% RSLogix 500 project PROCESO.RSS, saved by version 8.40.00.08 %
PROJECT "UNTITLED"    % processor: MicroLogix 1500 %

PROGRAM FILES
  LAD 2   34 rungs

DATA FILES
  O0 OUTPUT  6 elements
  I1 INPUT  5 elements
  S2 STATUS  66 elements
  B3 BINARY  1 elements
  T4 TIMER  10 elements
  C5 COUNTER  1 elements
  R6 CONTROL  1 elements
  N7 INTEGER  1 elements
  F8 FLOAT  1 elements

LADDER 2
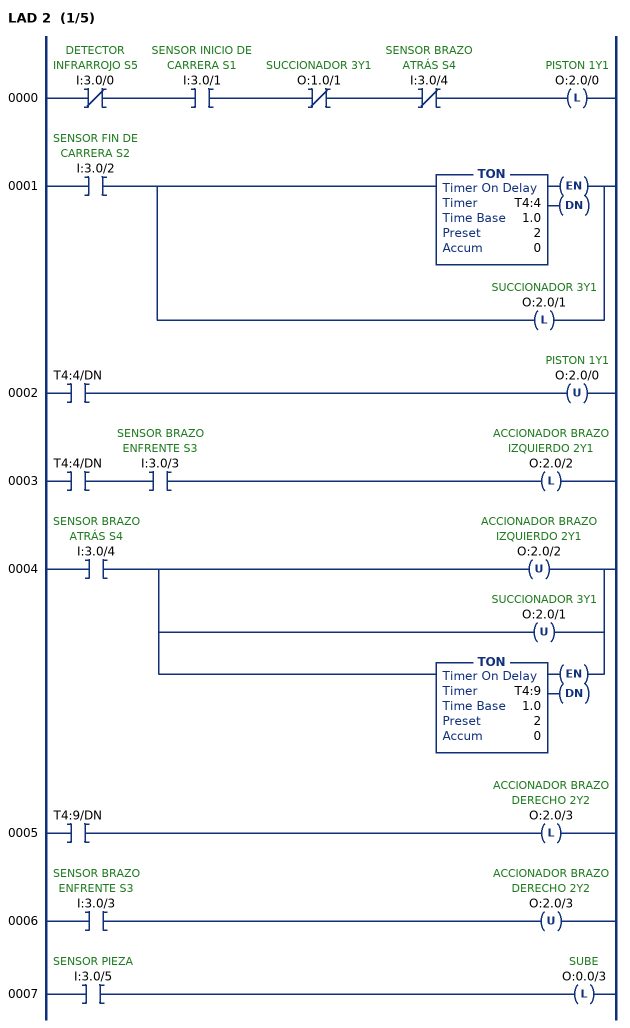
% Rung: 0 %
SOR XIO I:3.0/0 XIC I:3.0/1 XIO O:1.0/1 XIO I:3.0/4 OTL O:2.0/0 EOR
%   I:3.0/0  "DETECTOR INFRARROJO S5" %
%   I:3.0/1  "SENSOR INICIO DE CARRERA S1" %
%   O:1.0/1  "SUCCIONADOR 3Y1" %
%   I:3.0/4  "SENSOR BRAZO ATRÁS S4" %
%   O:2.0/0  "PISTON 1Y1" %
% Rung: 1 %
SOR XIC I:3.0/2 BST TON T4:4 1.0 2 0 NXB OTL O:2.0/1 BND EOR
%   I:3.0/2  "SENSOR FIN DE CARRERA S2" %
%   O:2.0/1  "SUCCIONADOR 3Y1" %
% Rung: 2 %
SOR XIC T4:4/DN OTU O:2.0/0 EOR
%   O:2.0/0  "PISTON 1Y1" %
% Rung: 3 %
SOR XIC T4:4/DN XIC I:3.0/3 OTL O:2.0/2 EOR
%   I:3.0/3  "SENSOR BRAZO ENFRENTE S3" %
%   O:2.0/2  "ACCIONADOR BRAZO IZQUIERDO 2Y1" %
% Rung: 4 %
SOR XIC I:3.0/4 BST OTU O:2.0/2 NXB BST OTU O:2.0/1 NXB TON T4:9 1.0 2 0 BND BND EOR
%   I:3.0/4  "SENSOR BRAZO ATRÁS S4" %
%   O:2.0/2  "ACCIONADOR BRAZO IZQUIERDO 2Y1" %
%   O:2.0/1  "SUCCIONADOR 3Y1" %
% Rung: 5 %
SOR XIC T4:9/DN OTL O:2.0/3 EOR
%   O:2.0/3  "ACCIONADOR BRAZO DERECHO 2Y2" %
% Rung: 6 %
SOR XIC I:3.0/3 OTU O:2.0/3 EOR
%   I:3.0/3  "SENSOR BRAZO ENFRENTE S3" %
%   O:2.0/3  "ACCIONADOR BRAZO DERECHO 2Y2" %
% Rung: 7 %
SOR XIC I:3.0/5 OTL O:0.0/3 EOR
%   I:3.0/5  "SENSOR PIEZA" %
%   O:0.0/3  "SUBE" %

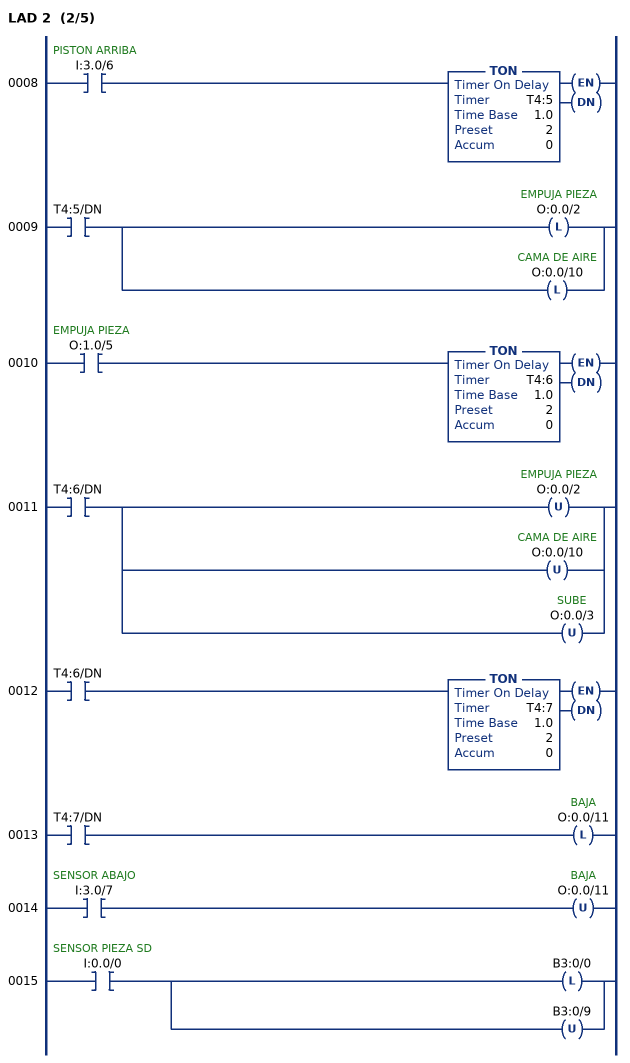
% Rung: 8 %
SOR XIC I:3.0/6 TON T4:5 1.0 2 0 EOR
%   I:3.0/6  "PISTON ARRIBA" %
% Rung: 9 %
SOR XIC T4:5/DN BST OTL O:0.0/2 NXB OTL O:0.0/10 BND EOR
%   O:0.0/2  "EMPUJA PIEZA" %
%   O:0.0/10  "CAMA DE AIRE" %
% Rung: 10 %
SOR XIC O:1.0/5 TON T4:6 1.0 2 0 EOR
%   O:1.0/5  "EMPUJA PIEZA" %
% Rung: 11 %
SOR XIC T4:6/DN BST OTU O:0.0/2 NXB BST OTU O:0.0/10 NXB OTU O:0.0/3 BND BND EOR
%   O:0.0/2  "EMPUJA PIEZA" %
%   O:0.0/10  "CAMA DE AIRE" %
%   O:0.0/3  "SUBE" %
% Rung: 12 %
SOR XIC T4:6/DN TON T4:7 1.0 2 0 EOR
% Rung: 13 %
SOR XIC T4:7/DN OTL O:0.0/11 EOR
%   O:0.0/11  "BAJA" %
% Rung: 14 %
SOR XIC I:3.0/7 OTU O:0.0/11 EOR
%   I:3.0/7  "SENSOR ABAJO" %
%   O:0.0/11  "BAJA" %
% Rung: 15 %
SOR XIC I:0.0/0 BST OTL B3:0/0 NXB OTU B3:0/9 BND EOR
%   I:0.0/0  "SENSOR PIEZA SD" %

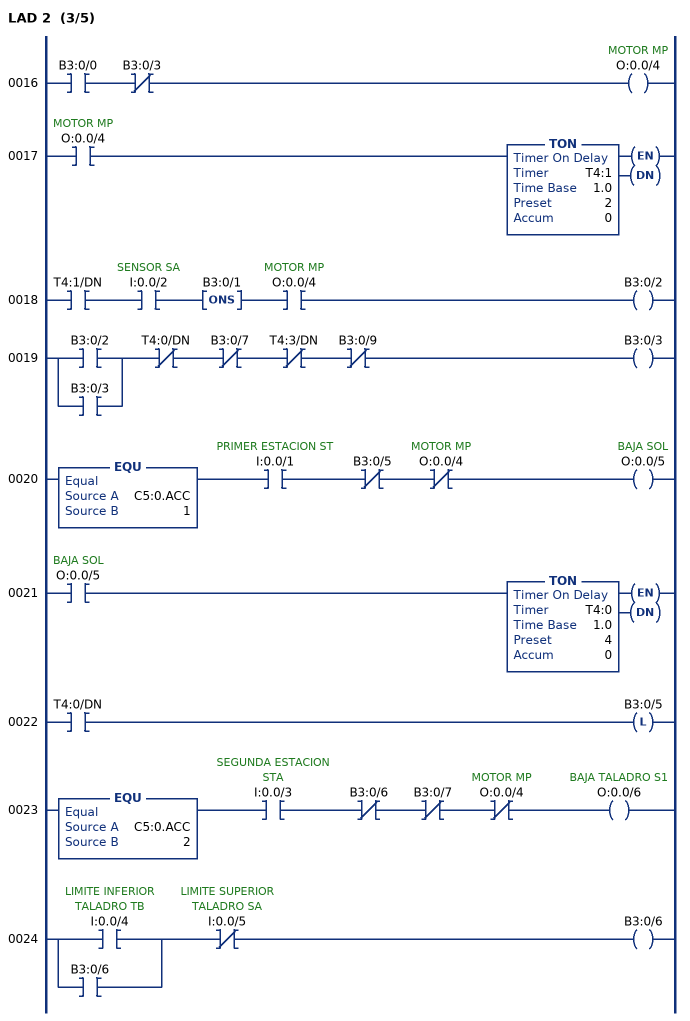
% Rung: 16 %
SOR XIC B3:0/0 XIO B3:0/3 OTE O:0.0/4 EOR
%   O:0.0/4  "MOTOR MP" %
% Rung: 17 %
SOR XIC O:0.0/4 TON T4:1 1.0 2 0 EOR
%   O:0.0/4  "MOTOR MP" %
% Rung: 18 %
SOR XIC T4:1/DN XIC I:0.0/2 ONS B3:0/1 XIC O:0.0/4 OTE B3:0/2 EOR
%   I:0.0/2  "SENSOR SA" %
%   O:0.0/4  "MOTOR MP" %
% Rung: 19 %
SOR BST XIC B3:0/2 NXB XIC B3:0/3 BND XIO T4:0/DN XIO B3:0/7 XIO T4:3/DN XIO B3:0/9 OTE B3:0/3 EOR
% Rung: 20 %
SOR EQU C5:0.ACC 1 XIC I:0.0/1 XIO B3:0/5 XIO O:0.0/4 OTE O:0.0/5 EOR
%   I:0.0/1  "PRIMER ESTACION ST" %
%   O:0.0/4  "MOTOR MP" %
%   O:0.0/5  "BAJA SOL" %
% Rung: 21 %
SOR XIC O:0.0/5 TON T4:0 1.0 4 0 EOR
%   O:0.0/5  "BAJA SOL" %
% Rung: 22 %
SOR XIC T4:0/DN OTL B3:0/5 EOR
% Rung: 23 %
SOR EQU C5:0.ACC 2 XIC I:0.0/3 XIO B3:0/6 XIO B3:0/7 XIO O:0.0/4 OTE O:0.0/6 EOR
%   I:0.0/3  "SEGUNDA ESTACION STA" %
%   O:0.0/4  "MOTOR MP" %
%   O:0.0/6  "BAJA TALADRO S1" %
% Rung: 24 %
SOR BST XIC I:0.0/4 NXB XIC B3:0/6 BND XIO I:0.0/5 OTE B3:0/6 EOR
%   I:0.0/4  "LIMITE INFERIOR TALADRO TB" %
%   I:0.0/5  "LIMITE SUPERIOR TALADRO SA" %

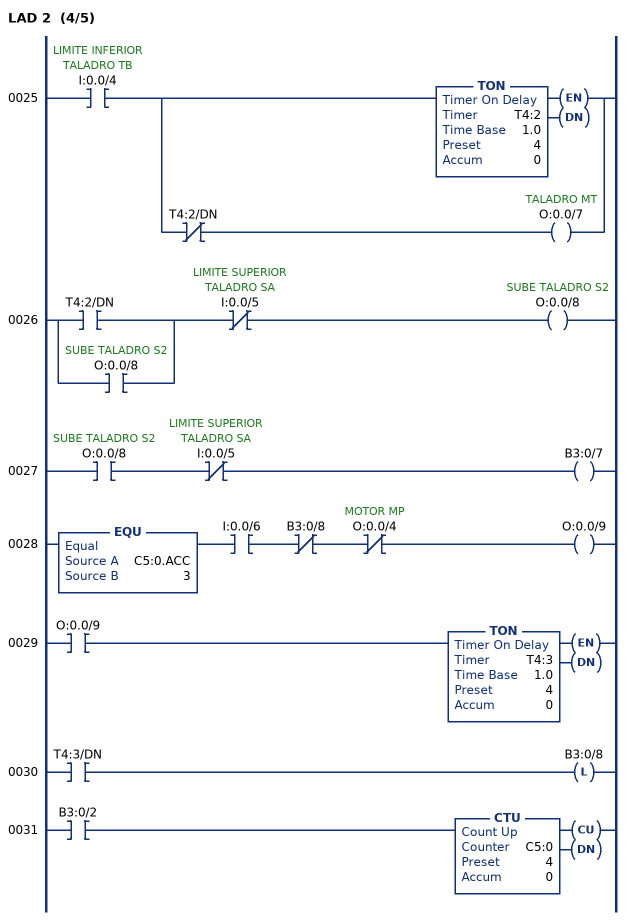
% Rung: 25 %
SOR XIC I:0.0/4 BST TON T4:2 1.0 4 0 NXB XIO T4:2/DN OTE O:0.0/7 BND EOR
%   I:0.0/4  "LIMITE INFERIOR TALADRO TB" %
%   O:0.0/7  "TALADRO MT" %
% Rung: 26 %
SOR BST XIC T4:2/DN NXB XIC O:0.0/8 BND XIO I:0.0/5 OTE O:0.0/8 EOR
%   O:0.0/8  "SUBE TALADRO S2" %
%   I:0.0/5  "LIMITE SUPERIOR TALADRO SA" %
% Rung: 27 %
SOR XIC O:0.0/8 XIO I:0.0/5 OTE B3:0/7 EOR
%   O:0.0/8  "SUBE TALADRO S2" %
%   I:0.0/5  "LIMITE SUPERIOR TALADRO SA" %
% Rung: 28 %
SOR EQU C5:0.ACC 3 XIC I:0.0/6 XIO B3:0/8 XIO O:0.0/4 OTE O:0.0/9 EOR
%   O:0.0/4  "MOTOR MP" %
% Rung: 29 %
SOR XIC O:0.0/9 TON T4:3 1.0 4 0 EOR
% Rung: 30 %
SOR XIC T4:3/DN OTL B3:0/8 EOR
% Rung: 31 %
SOR XIC B3:0/2 CTU C5:0 4 0 EOR

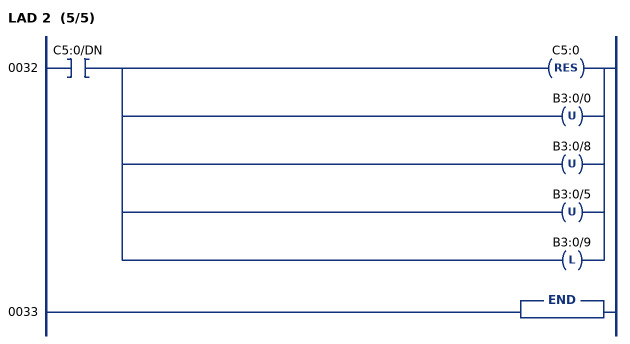
% Rung: 32 %
SOR XIC C5:0/DN BST RES C5:0 NXB BST OTU B3:0/0 NXB BST OTU B3:0/8 NXB BST OTU B3:0/5 NXB OTL B3:0/9 BND BND BND BND EOR
% Rung: 33 %
SOR END EOR

OTHER DOCUMENTED ADDRESSES
  O:1.0/0  "PISTON 1Y1"
  O:1.0/2  "ACCIONADOR BRAZO IZQUIERDO 2Y1"
  O:1.0/3  "ACCIONADOR BRAZO DERECHO 2Y2"
  O:1.0/4  "SUBE"
  O:1.0/6  "CAMA DE AIRE"
  O:1.0/7  "BAJA"
  O:2.0/4  "SUBE"
  O:2.0/5  "EMPUJA PIEZA"
  O:2.0/6  "CAMA DE AIRE"
  O:2.0/7  "BAJA"

DATA TABLE (non-zero values as saved)
DATA T4
% .PRE .ACC %
% T4:0 % 4 0
% T4:1 % 2 0
% T4:2 % 4 0
% T4:3 % 4 0
% T4:4 % 2 0
% T4:5 % 2 0
% T4:6 % 2 0
% T4:7 % 2 0
% T4:9 % 2 0
DATA C5
% .PRE .ACC %
% C5:0 % 4 0
